Fanuc KAREL source: KS00014.KL

PROGRAM KS00014
%NOLOCKGROUP
TYPE
  REC_T = STRUCTURE
    VALUE: INTEGER
    FLAG: BOOLEAN
  ENDSTRUCTURE
VAR
  A: PATH
  B: PATH
  FLAG: BOOLEAN
  N: INTEGER
  STATUS: INTEGER
  PN: STRING[80]
  VN: STRING[80]
BEGIN
  PN = ''
  VN = 'A'
  SET_VAR(N, PN, VN, A, STATUS)
END KS00014
